// TIA Portal V20 export
// export: Created 2025-12-01T14:57:43.3268594Z, ExportSetting None, DisplayName Totally Integrated Automation Portal, DisplayVersion V20 Update 3, DisplayName TIA Portal Openness, DisplayVersion V20 Update 3, DisplayName TIA Portal Version Control Interface, DisplayVersion V20 Update 3, DisplayName STEP 7 Professional, DisplayVersion V20 Update 3, DisplayName STEP 7 Safety, DisplayVersion V20 Update 2, DisplayName WinCC Basic/Comfort/Advanced, DisplayVersion V20 Update 3, DisplayName WinCC Professional, DisplayVersion V20 Update 3, DisplayName WinCC Unified, DisplayVersion V20 Update 3
FUNCTION "FC499_Mirar_Estado_Vacio" : Void   // FC499, LAD
{ S7_Optimized_Access := 'FALSE' }
AUTHOR : TLigero
NAME : 20150226
VERSION : 3.0
// stored: AutoNumber false, SetENOAutomatically false
   VAR_INPUT
      Numero_Mesa_Ini : UInt;
      Numero_Mesa_Fin : UInt;
   END_VAR
   VAR_OUTPUT
      Mesas_Vacias : Bool;
   END_VAR
   VAR_TEMP
      Aux_contador : UInt;
   END_VAR
BEGIN

REGION Network 1 (SCL)
   FOR #Aux_contador := #Numero_Mesa_Ini TO #Numero_Mesa_Fin DO
       IF "DB900_Estado_Mesas".EstadoVI[#Aux_contador].Etapa_Vacia = false THEN
           #Mesas_Vacias := FALSE;
           RETURN;
       END_IF;
   END_FOR;
   #Mesas_Vacias := true;
END_REGION
END_FUNCTION
